// TIA Portal project "ElevatorController" (V14)

(* hardware
DEVICE "S7-1200 station_1"  S7-1200 Station
   slot 0: "Rack_0"  S7-1200 Rack  Rack  V1.0
   slot 1: "PLC_1"  CPU 1214C DC/DC/DC  6ES7 214-1AE30-0XB0  V2.2
   slot 101: "CM 1243-5"  CM 1243-5  6GK7 243-5DX30-0XE0  V1.0
DEVICE "GSD device_1"  GSD.Device
   slot 0: "机架_0"  Rail
   slot 0: "Slave_1"  PM125  V2.0
DEVICE "DESKTOP-VBI98IE"  SIMATIC PC station
   slot 0: "SIMATIC PC station"  Rail  SIMATIC PC-Station  V1.0
      slot 125: "Stationmanager"  Station_Manager  V6.0.4
   slot 1: "HMI_RT_1"  WinCC RT Advanced  6AV2 104-0xxxx-xxxx  14.0.1.0
      slot 33792: "主机接口"  Host interface
   slot 2: "IE general_1"  IE General  IE_CP  V8.2.0
*)

// ===== PLC "PLC_1"  CPU 1214C DC/DC/DC =====

VAR_GLOBAL   // PLC tag table "默认变量表"
   "X0" AT %I0.0 : Bool;   // 一层到层开关
   "X1" AT %I0.1 : Bool;   // 二层到层开关
   "X2" AT %I0.2 : Bool;   // 三层到层开关
   "X3" AT %I0.3 : Bool;   // 四层到层开关
   "X4" AT %I0.4 : Bool;   // 一层呼叫按钮
   "X5" AT %I0.5 : Bool;   // 二层呼叫按钮
   "X6" AT %I0.6 : Bool;   // 三层呼叫按钮
   "X7" AT %I0.7 : Bool;   // 四层呼叫按钮
   "X8" AT %I1.0 : Bool;
   "X9" AT %I1.1 : Bool;
   "X10" AT %I1.2 : Bool;
   "X11" AT %I1.3 : Bool;
   "Y0" AT %Q1.4 : Bool;   // 数码管A
   "Y1" AT %Q1.5 : Bool;   // 数码管B
   "Y2" AT %Q1.6 : Bool;   // 数码管C
   "Y3" AT %Q1.7 : Bool;   // 数码管D
   "Y4" AT %Q2.0 : Bool;   // 数码管E
   "Y5" AT %Q2.1 : Bool;   // 数码管F
   "Y6" AT %Q2.2 : Bool;   // 数码管G
   "Y7" AT %Q2.3 : Bool;
   "Y8" AT %Q2.4 : Bool;
   "Y9" AT %Q2.5 : Bool;
   "Y10" AT %Q2.6 : Bool;   // 电梯向上运行
   "Y11" AT %Q2.7 : Bool;   // 电梯向下运行
   "Y12" AT %Q3.0 : Bool;   // 一层向上呼叫指示灯
   "Y13" AT %Q3.1 : Bool;   // 二层向上呼叫指示灯
   "Y14" AT %Q3.2 : Bool;   // 三层向上呼叫指示灯
   "Y17" AT %Q3.3 : Bool;   // 二层向下呼叫指示灯
   "S13" AT %M0.0 : Bool;
   "S12" AT %M0.1 : Bool;
   "S11" AT %M0.2 : Bool;
   "R1" AT %M0.3 : Bool;
   "S14" AT %M0.4 : Bool;
   "Y15" AT %M0.5 : Bool;   // 四层向下呼叫指示
   "Y16" AT %M0.6 : Bool;   // 三层向下呼叫指示
   "S1" AT %M0.7 : Bool;
   "S2" AT %M1.0 : Bool;
   "S3" AT %M1.1 : Bool;
   "S4" AT %M1.2 : Bool;
   "T1" AT %M1.3 : Bool;
   "M0" AT %M1.4 : Bool;   // 电机
   "M1" AT %M1.5 : Bool;
   "M2" AT %M1.6 : Bool;
   "Tag_1" AT %MB400 : Byte;
   "Tag_2" AT %QB2 : Byte;
   "Tag_3" AT %QB3 : Byte;
   "Tag_4" AT %MB2 : Byte;
END_VAR

TYPE "用户数据类型_1"
   STRUCT
      "Struct" : Struct
      END_STRUCT;
   END_STRUCT;
END_TYPE

DATA_BLOCK "输出变量"   // DB1
{ S7_Optimized_Access := 'FALSE' }
VERSION : 0.1
   VAR
      "1层上行呼梯按钮指示灯" : Bool;
      "2层上行呼梯按钮指示灯" : Bool;
      "3层上行呼梯按钮指示灯" : Bool;
      "4层上行呼梯按钮指示灯" : Bool;
      "5层上行呼梯按钮指示灯" : Bool;
      "6层上行呼梯按钮指示灯" : Bool;
      "7层上行呼梯按钮指示灯" : Bool;
      "8层上行呼梯按钮指示灯" : Bool;
      "9层上行呼梯按钮指示灯" : Bool;
      "2层下行呼梯按钮指示灯" : Bool;
      "3层下行呼梯按钮指示灯" : Bool;
      "4层下行呼梯按钮指示灯" : Bool;
      "5层下行呼梯按钮指示灯" : Bool;
      "6层下行呼梯按钮指示灯" : Bool;
      "7层下行呼梯按钮指示灯" : Bool;
      "8层下行呼梯按钮指示灯" : Bool;
      "9层下行呼梯按钮指示灯" : Bool;
      "10层下行呼梯按钮指示灯" : Bool;
      "1号梯1层按钮指示灯" : Bool;
      "1号梯2层按钮指示灯" : Bool;
      "1号梯3层按钮指示灯" : Bool;
      "1号梯4层按钮指示灯" : Bool;
      "1号梯5层按钮指示灯" : Bool;
      "1号梯6层按钮指示灯" : Bool;
      "1号梯7层按钮指示灯" : Bool;
      "1号梯8层按钮指示灯" : Bool;
      "1号梯9层按钮指示灯" : Bool;
      "1号梯10层按钮指示灯" : Bool;
      "1号梯LEDa" : Bool;
      "1号梯LEDb" : Bool;
      "1号梯LEDc" : Bool;
      "1号梯LEDd" : Bool;
      "1号梯LEDe" : Bool;
      "1号梯LEDf" : Bool;
      "1号梯LEDg" : Bool;
      "1号梯LEDh" : Bool;
      "1号梯LEDi" : Bool;
      "1号梯LEDj" : Bool;
      "1号梯LEDk" : Bool;
      "1号梯LEDl" : Bool;
      "1号梯LEDm" : Bool;
      "1号梯LEDn" : Bool;
      "1号梯上行指示" : Bool;
      "1号梯下行指示" : Bool;
      "1号梯故障指示" : Bool;
      "1号梯照明指示" : Bool;
      "1号梯风扇指示" : Bool;
      "1号梯满载指示" : Bool;
      "1号梯电机启动信号" : Bool;
      "1号梯上行接触器" : Bool;
      "1号梯下行接触器" : Bool;
      "1号梯高速接触器" : Bool;
      "1号梯低速接触器" : Bool;
      "1号梯开门继电器" : Bool;
      "1号梯关门继电器" : Bool;
      "1号梯1级减速制动" : Bool;
      "1号梯2级减速制动" : Bool;
      "1号梯3级减速制动" : Bool;
      "2号梯1层按钮指示灯" : Bool;
      "2号梯2层按钮指示灯" : Bool;
      "2号梯3层按钮指示灯" : Bool;
      "2号梯4层按钮指示灯" : Bool;
      "2号梯5层按钮指示灯" : Bool;
      "2号梯6层按钮指示灯" : Bool;
      "2号梯7层按钮指示灯" : Bool;
      "2号梯8层按钮指示灯" : Bool;
      "2号梯9层按钮指示灯" : Bool;
      "2号梯10层按钮指示灯" : Bool;
      "2号梯LEDa" : Bool;
      "2号梯LEDb" : Bool;
      "2号梯LEDc" : Bool;
      "2号梯LEDd" : Bool;
      "2号梯LEDe" : Bool;
      "2号梯LEDf" : Bool;
      "2号梯LEDg" : Bool;
      "2号梯LEDh" : Bool;
      "2号梯LEDi" : Bool;
      "2号梯LEDj" : Bool;
      "2号梯LEDk" : Bool;
      "2号梯LEDl" : Bool;
      "2号梯LEDm" : Bool;
      "2号梯LEDn" : Bool;
      "2号梯上行指示" : Bool;
      "2号梯下行指示" : Bool;
      "2号梯故障指示" : Bool;
      "2号梯照明指示" : Bool;
      "2号梯风扇指示" : Bool;
      "2号梯满载指示" : Bool;
      "2号梯电机启动信号" : Bool;
      "2号梯上行接触器" : Bool;
      "2号梯下行接触器" : Bool;
      "2号梯高速接触器" : Bool;
      "2号梯低速接触器" : Bool;
      "2号梯开门继电器" : Bool;
      "2号梯关门继电器" : Bool;
      "2号梯1级减速制动" : Bool;
      "2号梯2级减速制动" : Bool;
      "2号梯3级减速制动" : Bool;
      "3号梯1层按钮指示灯" : Bool;
      "3号梯2层按钮指示灯" : Bool;
      "3号梯3层按钮指示灯" : Bool;
      "3号梯4层按钮指示灯" : Bool;
      "3号梯5层按钮指示灯" : Bool;
      "3号梯6层按钮指示灯" : Bool;
      "3号梯7层按钮指示灯" : Bool;
      "3号梯8层按钮指示灯" : Bool;
      "3号梯9层按钮指示灯" : Bool;
      "3号梯10层按钮指示灯" : Bool;
      "3号梯LEDa" : Bool;
      "3号梯LEDb" : Bool;
      "3号梯LEDc" : Bool;
      "3号梯LEDd" : Bool;
      "3号梯LEDe" : Bool;
      "3号梯LEDf" : Bool;
      "3号梯LEDg" : Bool;
      "3号梯LEDh" : Bool;
      "3号梯LEDi" : Bool;
      "3号梯LEDj" : Bool;
      "3号梯LEDk" : Bool;
      "3号梯LEDl" : Bool;
      "3号梯LEDm" : Bool;
      "3号梯LEDn" : Bool;
      "3号梯上行指示" : Bool;
      "3号梯下行指示" : Bool;
      "3号梯故障指示" : Bool;
      "3号梯照明指示" : Bool;
      "3号梯风扇指示" : Bool;
      "3号梯满载指示" : Bool;
      "3号梯电机启动信号" : Bool;
      "3号梯上行接触器" : Bool;
      "3号梯下行接触器" : Bool;
      "3号梯高速接触器" : Bool;
      "3号梯低速接触器" : Bool;
      "3号梯开门继电器" : Bool;
      "3号梯关门继电器" : Bool;
      "3号梯1级减速制动" : Bool;
      "3号梯2级减速制动" : Bool;
      "3号梯3级减速制动" : Bool;
      "4号梯1层按钮指示灯" : Bool;
      "4号梯2层按钮指示灯" : Bool;
      "4号梯3层按钮指示灯" : Bool;
      "4号梯4层按钮指示灯" : Bool;
      "4号梯5层按钮指示灯" : Bool;
      "4号梯6层按钮指示灯" : Bool;
      "4号梯7层按钮指示灯" : Bool;
      "4号梯8层按钮指示灯" : Bool;
      "4号梯9层按钮指示灯" : Bool;
      "4号梯10层按钮指示灯" : Bool;
      "4号梯LEDa" : Bool;
      "4号梯LEDb" : Bool;
      "4号梯LEDc" : Bool;
      "4号梯LEDd" : Bool;
      "4号梯LEDe" : Bool;
      "4号梯LEDf" : Bool;
      "4号梯LEDg" : Bool;
      "4号梯LEDh" : Bool;
      "4号梯LEDi" : Bool;
      "4号梯LEDj" : Bool;
      "4号梯LEDk" : Bool;
      "4号梯LEDl" : Bool;
      "4号梯LEDm" : Bool;
      "4号梯LEDn" : Bool;
      "4号梯上行指示" : Bool;
      "4号梯下行指示" : Bool;
      "4号梯故障指示" : Bool;
      "4号梯照明指示" : Bool;
      "4号梯风扇指示" : Bool;
      "4号梯满载指示" : Bool;
      "4号梯电机启动信号" : Bool;
      "4号梯上行接触器" : Bool;
      "4号梯下行接触器" : Bool;
      "4号梯高速接触器" : Bool;
      "4号梯低速接触器" : Bool;
      "4号梯开门继电器" : Bool;
      "4号梯关门继电器" : Bool;
      "4号梯1级减速制动" : Bool;
      "4号梯2级减速制动" : Bool;
      "4号梯3级减速制动" : Bool;
      "5号梯1层按钮指示灯" : Bool;
      "5号梯2层按钮指示灯" : Bool;
      "5号梯3层按钮指示灯" : Bool;
      "5号梯4层按钮指示灯" : Bool;
      "5号梯5层按钮指示灯" : Bool;
      "5号梯6层按钮指示灯" : Bool;
      "5号梯7层按钮指示灯" : Bool;
      "5号梯8层按钮指示灯" : Bool;
      "5号梯9层按钮指示灯" : Bool;
      "5号梯10层按钮指示灯" : Bool;
      "5号梯LEDa" : Bool;
      "5号梯LEDb" : Bool;
      "5号梯LEDc" : Bool;
      "5号梯LEDd" : Bool;
      "5号梯LEDe" : Bool;
      "5号梯LEDf" : Bool;
      "5号梯LEDg" : Bool;
      "5号梯LEDh" : Bool;
      "5号梯LEDi" : Bool;
      "5号梯LEDj" : Bool;
      "5号梯LEDk" : Bool;
      "5号梯LEDl" : Bool;
      "5号梯LEDm" : Bool;
      "5号梯LEDn" : Bool;
      "5号梯上行指示" : Bool;
      "5号梯下行指示" : Bool;
      "5号梯故障指示" : Bool;
      "5号梯照明指示" : Bool;
      "5号梯风扇指示" : Bool;
      "5号梯满载指示" : Bool;
      "5号梯电机启动信号" : Bool;
      "5号梯上行接触器" : Bool;
      "5号梯下行接触器" : Bool;
      "5号梯高速接触器" : Bool;
      "5号梯低速接触器" : Bool;
      "5号梯开门继电器" : Bool;
      "5号梯关门继电器" : Bool;
      "5号梯1级减速制动" : Bool;
      "5号梯2级减速制动" : Bool;
      "5号梯3级减速制动" : Bool;
      "6号梯1层按钮指示灯" : Bool;
      "6号梯2层按钮指示灯" : Bool;
      "6号梯3层按钮指示灯" : Bool;
      "6号梯4层按钮指示灯" : Bool;
      "6号梯5层按钮指示灯" : Bool;
      "6号梯6层按钮指示灯" : Bool;
      "6号梯7层按钮指示灯" : Bool;
      "6号梯8层按钮指示灯" : Bool;
      "6号梯9层按钮指示灯" : Bool;
      "6号梯10层按钮指示灯" : Bool;
      "6号梯LEDa" : Bool;
      "6号梯LEDb" : Bool;
      "6号梯LEDc" : Bool;
      "6号梯LEDd" : Bool;
      "6号梯LEDe" : Bool;
      "6号梯LEDf" : Bool;
      "6号梯LEDg" : Bool;
      "6号梯LEDh" : Bool;
      "6号梯LEDi" : Bool;
      "6号梯LEDj" : Bool;
      "6号梯LEDk" : Bool;
      "6号梯LEDl" : Bool;
      "6号梯LEDm" : Bool;
      "6号梯LEDn" : Bool;
      "6号梯上行指示" : Bool;
      "6号梯下行指示" : Bool;
      "6号梯故障指示" : Bool;
      "6号梯照明指示" : Bool;
      "6号梯风扇指示" : Bool;
      "6号梯满载指示" : Bool;
      "6号梯电机启动信号" : Bool;
      "6号梯上行接触器" : Bool;
      "6号梯下行接触器" : Bool;
      "6号梯高速接触器" : Bool;
      "6号梯低速接触器" : Bool;
      "6号梯开门继电器" : Bool;
      "6号梯关门继电器" : Bool;
      "6号梯1级减速制动" : Bool;
      "6号梯2级减速制动" : Bool;
      "6号梯3级减速制动" : Bool;
      准备就绪信号 : Bool;
   END_VAR
BEGIN
END_DATA_BLOCK

DATA_BLOCK "输入变量"   // DB2
{ S7_Optimized_Access := 'FALSE' }
VERSION : 0.1
   VAR
      "1层上行呼梯按钮" : Bool;
      "2层上行呼梯按钮" : Bool;
      "3层上行呼梯按钮" : Bool;
      "4层上行呼梯按钮" : Bool;
      "5层上行呼梯按钮" : Bool;
      "6层上行呼梯按钮" : Bool;
      "7层上行呼梯按钮" : Bool;
      "8层上行呼梯按钮" : Bool;
      "9层上行呼梯按钮" : Bool;
      "2层下行呼梯按钮" : Bool;
      "3层下行呼梯按钮" : Bool;
      "4层下行呼梯按钮" : Bool;
      "5层下行呼梯按钮" : Bool;
      "6层下行呼梯按钮" : Bool;
      "7层下行呼梯按钮" : Bool;
      "8层下行呼梯按钮" : Bool;
      "9层下行呼梯按钮" : Bool;
      "10层下行呼梯按钮" : Bool;
      "1号梯轿内选层按钮1" : Bool;
      "1号梯轿内选层按钮2" : Bool;
      "1号梯轿内选层按钮3" : Bool;
      "1号梯轿内选层按钮4" : Bool;
      "1号梯轿内选层按钮5" : Bool;
      "1号梯轿内选层按钮6" : Bool;
      "1号梯轿内选层按钮7" : Bool;
      "1号梯轿内选层按钮8" : Bool;
      "1号梯轿内选层按钮9" : Bool;
      "1号梯轿内选层按钮10" : Bool;
      "1号梯轿内开门按钮" : Bool;
      "1号梯轿内关门按钮" : Bool;
      "1号梯光幕信号" : Bool;
      "1号梯超重信号" : Bool;
      "1号梯检修信号" : Bool;
      "1号梯轿厢门锁信号" : Bool;
      "1号梯1楼层门锁信号" : Bool;
      "1号梯2楼层门锁信号" : Bool;
      "1号梯3楼层门锁信号" : Bool;
      "1号梯4楼层门锁信号" : Bool;
      "1号梯5楼层门锁信号" : Bool;
      "1号梯6楼层门锁信号" : Bool;
      "1号梯7楼层门锁信号" : Bool;
      "1号梯8楼层门锁信号" : Bool;
      "1号梯9楼层门锁信号" : Bool;
      "1号梯10楼层门锁信号" : Bool;
      "1号梯开门到位" : Bool;
      "1号梯关门到位" : Bool;
      "1号梯上平层信号" : Bool;
      "1号梯下平层信号" : Bool;
      "1号梯上端站第1限位" : Bool;
      "1号梯上端站第2限位" : Bool;
      "1号梯下端站第1限位" : Bool;
      "1号梯下端站第2限位" : Bool;
      "2号梯轿内选层按钮1" : Bool;
      "2号梯轿内选层按钮2" : Bool;
      "2号梯轿内选层按钮3" : Bool;
      "2号梯轿内选层按钮4" : Bool;
      "2号梯轿内选层按钮5" : Bool;
      "2号梯轿内选层按钮6" : Bool;
      "2号梯轿内选层按钮7" : Bool;
      "2号梯轿内选层按钮8" : Bool;
      "2号梯轿内选层按钮9" : Bool;
      "2号梯轿内选层按钮10" : Bool;
      "2号梯轿内开门按钮" : Bool;
      "2号梯轿内关门按钮" : Bool;
      "2号梯光幕信号" : Bool;
      "2号梯超重信号" : Bool;
      "2号梯检修信号" : Bool;
      "2号梯轿厢门锁信号" : Bool;
      "2号梯1楼层门锁信号" : Bool;
      "2号梯2楼层门锁信号" : Bool;
      "2号梯3楼层门锁信号" : Bool;
      "2号梯4楼层门锁信号" : Bool;
      "2号梯5楼层门锁信号" : Bool;
      "2号梯6楼层门锁信号" : Bool;
      "2号梯7楼层门锁信号" : Bool;
      "2号梯8楼层门锁信号" : Bool;
      "2号梯9楼层门锁信号" : Bool;
      "2号梯10楼层门锁信号" : Bool;
      "2号梯开门到位" : Bool;
      "2号梯关门到位" : Bool;
      "2号梯上平层信号" : Bool;
      "2号梯下平层信号" : Bool;
      "2号梯上端站第1限位" : Bool;
      "2号梯上端站第2限位" : Bool;
      "2号梯下端站第1限位" : Bool;
      "2号梯下端站第2限位" : Bool;
      "3号梯轿内选层按钮1" : Bool;
      "3号梯轿内选层按钮2" : Bool;
      "3号梯轿内选层按钮3" : Bool;
      "3号梯轿内选层按钮4" : Bool;
      "3号梯轿内选层按钮5" : Bool;
      "3号梯轿内选层按钮6" : Bool;
      "3号梯轿内选层按钮7" : Bool;
      "3号梯轿内选层按钮8" : Bool;
      "3号梯轿内选层按钮9" : Bool;
      "3号梯轿内选层按钮10" : Bool;
      "3号梯轿内开门按钮" : Bool;
      "3号梯轿内关门按钮" : Bool;
      "3号梯光幕信号" : Bool;
      "3号梯超重信号" : Bool;
      "3号梯检修信号" : Bool;
      "3号梯轿厢门锁信号" : Bool;
      "3号梯1楼层门锁信号" : Bool;
      "3号梯2楼层门锁信号" : Bool;
      "3号梯3楼层门锁信号" : Bool;
      "3号梯4楼层门锁信号" : Bool;
      "3号梯5楼层门锁信号" : Bool;
      "3号梯6楼层门锁信号" : Bool;
      "3号梯7楼层门锁信号" : Bool;
      "3号梯8楼层门锁信号" : Bool;
      "3号梯9楼层门锁信号" : Bool;
      "3号梯10楼层门锁信号" : Bool;
      "3号梯开门到位" : Bool;
      "3号梯关门到位" : Bool;
      "3号梯上平层信号" : Bool;
      "3号梯下平层信号" : Bool;
      "3号梯上端站第1限位" : Bool;
      "3号梯上端站第2限位" : Bool;
      "3号梯下端站第1限位" : Bool;
      "3号梯下端站第2限位" : Bool;
      "4号梯轿内选层按钮1" : Bool;
      "4号梯轿内选层按钮2" : Bool;
      "4号梯轿内选层按钮3" : Bool;
      "4号梯轿内选层按钮4" : Bool;
      "4号梯轿内选层按钮5" : Bool;
      "4号梯轿内选层按钮6" : Bool;
      "4号梯轿内选层按钮7" : Bool;
      "4号梯轿内选层按钮8" : Bool;
      "4号梯轿内选层按钮9" : Bool;
      "4号梯轿内选层按钮10" : Bool;
      "4号梯轿内开门按钮" : Bool;
      "4号梯轿内关门按钮" : Bool;
      "4号梯光幕信号" : Bool;
      "4号梯超重信号" : Bool;
      "4号梯检修信号" : Bool;
      "4号梯轿厢门锁信号" : Bool;
      "4号梯1楼层门锁信号" : Bool;
      "4号梯2楼层门锁信号" : Bool;
      "4号梯3楼层门锁信号" : Bool;
      "4号梯4楼层门锁信号" : Bool;
      "4号梯5楼层门锁信号" : Bool;
      "4号梯6楼层门锁信号" : Bool;
      "4号梯7楼层门锁信号" : Bool;
      "4号梯8楼层门锁信号" : Bool;
      "4号梯9楼层门锁信号" : Bool;
      "4号梯10楼层门锁信号" : Bool;
      "4号梯开门到位" : Bool;
      "4号梯关门到位" : Bool;
      "4号梯上平层信号" : Bool;
      "4号梯下平层信号" : Bool;
      "4号梯上端站第1限位" : Bool;
      "4号梯上端站第2限位" : Bool;
      "4号梯下端站第1限位" : Bool;
      "4号梯下端站第2限位" : Bool;
      "5号梯轿内选层按钮1" : Bool;
      "5号梯轿内选层按钮2" : Bool;
      "5号梯轿内选层按钮3" : Bool;
      "5号梯轿内选层按钮4" : Bool;
      "5号梯轿内选层按钮5" : Bool;
      "5号梯轿内选层按钮6" : Bool;
      "5号梯轿内选层按钮7" : Bool;
      "5号梯轿内选层按钮8" : Bool;
      "5号梯轿内选层按钮9" : Bool;
      "5号梯轿内选层按钮10" : Bool;
      "5号梯轿内开门按钮" : Bool;
      "5号梯轿内关门按钮" : Bool;
      "5号梯光幕信号" : Bool;
      "5号梯超重信号" : Bool;
      "5号梯检修信号" : Bool;
      "5号梯轿厢门锁信号" : Bool;
      "5号梯1楼层门锁信号" : Bool;
      "5号梯2楼层门锁信号" : Bool;
      "5号梯3楼层门锁信号" : Bool;
      "5号梯4楼层门锁信号" : Bool;
      "5号梯5楼层门锁信号" : Bool;
      "5号梯6楼层门锁信号" : Bool;
      "5号梯7楼层门锁信号" : Bool;
      "5号梯8楼层门锁信号" : Bool;
      "5号梯9楼层门锁信号" : Bool;
      "5号梯10楼层门锁信号" : Bool;
      "5号梯开门到位" : Bool;
      "5号梯关门到位" : Bool;
      "5号梯上平层信号" : Bool;
      "5号梯下平层信号" : Bool;
      "5号梯上端站第1限位" : Bool;
      "5号梯上端站第2限位" : Bool;
      "5号梯下端站第1限位" : Bool;
      "5号梯下端站第2限位" : Bool;
      "6号梯轿内选层按钮1" : Bool;
      "6号梯轿内选层按钮2" : Bool;
      "6号梯轿内选层按钮3" : Bool;
      "6号梯轿内选层按钮4" : Bool;
      "6号梯轿内选层按钮5" : Bool;
      "6号梯轿内选层按钮6" : Bool;
      "6号梯轿内选层按钮7" : Bool;
      "6号梯轿内选层按钮8" : Bool;
      "6号梯轿内选层按钮9" : Bool;
      "6号梯轿内选层按钮10" : Bool;
      "6号梯轿内开门按钮" : Bool;
      "6号梯轿内关门按钮" : Bool;
      "6号梯光幕信号" : Bool;
      "6号梯超重信号" : Bool;
      "6号梯检修信号" : Bool;
      "6号梯轿厢门锁信号" : Bool;
      "6号梯1楼层门锁信号" : Bool;
      "6号梯2楼层门锁信号" : Bool;
      "6号梯3楼层门锁信号" : Bool;
      "6号梯4楼层门锁信号" : Bool;
      "6号梯5楼层门锁信号" : Bool;
      "6号梯6楼层门锁信号" : Bool;
      "6号梯7楼层门锁信号" : Bool;
      "6号梯8楼层门锁信号" : Bool;
      "6号梯9楼层门锁信号" : Bool;
      "6号梯10楼层门锁信号" : Bool;
      "6号梯开门到位" : Bool;
      "6号梯关门到位" : Bool;
      "6号梯上平层信号" : Bool;
      "6号梯下平层信号" : Bool;
      "6号梯上端站第1限位" : Bool;
      "6号梯上端站第2限位" : Bool;
      "6号梯下端站第1限位" : Bool;
      "6号梯下端站第2限位" : Bool;
      自动运行信号 : Bool;
   END_VAR
BEGIN
END_DATA_BLOCK

ORGANIZATION_BLOCK "Main"   // OB1, LAD, ProgramCycle
TITLE = "Main Program Sweep (Cycle)"
{ S7_Optimized_Access := 'TRUE' }
VERSION : 0.1
   VAR_TEMP
      S14 : Bool;
      "”M0“" : Bool;
   END_VAR
BEGIN

REGION Network 1: 通讯输入
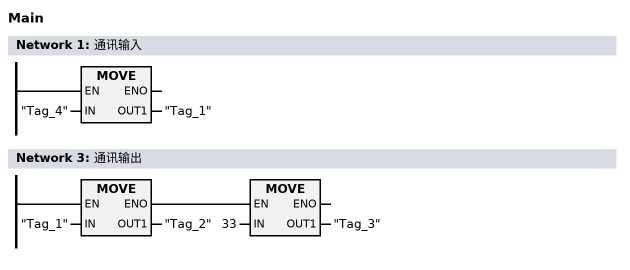
   RUNG wire#powerrail
      { S7_GenerateENO := "TRUE" } Move(in := "Tag_4", out1 => "Tag_1")
   END_RUNG
   // the same network as SCL:
   "Tag_1" := "Tag_4";
END_REGION

REGION Network 2: 主程序
END_REGION

REGION Network 3: 通讯输出
   RUNG wire#powerrail
      { S7_GenerateENO := "TRUE" } Move(in := "Tag_1", out1 => "Tag_2")
      { S7_GenerateENO := "TRUE" } Move(in := 33, out1 => "Tag_3")
   END_RUNG
   // the same network as SCL:
   // ENO of a box is taken as its EN; it also drops when the box reports an error
   "Tag_2" := "Tag_1";
   "Tag_3" := 33;
END_REGION
END_ORGANIZATION_BLOCK